FUNCTION_BLOCK POU
VAR_INPUT
END_VAR
VAR_OUTPUT
END_VAR
VAR
	CurrentState: MachineState;
	Lamp: BOOL;
END_VAR

IF CurrentState = off THEN 
	Lamp := FALSE; 
ELSIF CurrentState = On THEN 
	Lamp := TRUE; 
ELSIF CurrentState = Error THEN 
	//blink lamp
END_IF

END_FUNCTION_BLOCK

(* stored: Version 1.1.0.1
   POU POU: Id {5b40bf56-4e25-49bf-87c8-7c010d85423e}, SpecialFunc None *)
